Universal Robots URScript: 00B_04_Qu_BoXian.script

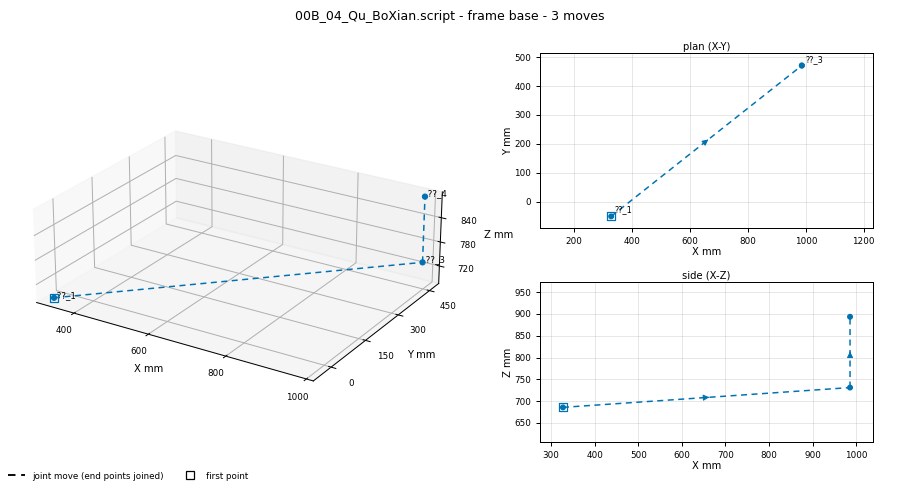
[picture p0: tool path of 00B_04_Qu_BoXian.script in frame base, 3 of 3 moves have a stored position in this frame; points joined in program order, loops and branches not executed]
def P00B_04_Qu_BoXian():
  set_gravity([0.0, 0.0, 9.82])
  set_safety_mode_transition_hardness(1)
  set_standard_analog_input_domain(0, 1)
  set_standard_analog_input_domain(1, 1)
  set_tool_analog_input_domain(0, 1)
  set_tool_analog_input_domain(1, 1)
  set_analog_outputdomain(0, 0)
  set_analog_outputdomain(1, 0)
  set_tool_voltage(24)
  set_input_actions_to_default()
  set_tcp(p[0.0,0.0,0.32,0.0,0.0,-0.5236])
  set_payload(8.0)
  global Zhua_1=[0.08063, -2.42649, -1.72682, -0.47876, 0.40808, -1.10831]
  global prepose=p[0.98979, -0.16931, -0.39963, 1.98720, 0.07234, 0.05469]
  global i_var_2=0
  global i_var_1=True
  global pose=p[0.98979, -0.31931, -0.39963, 1.98720, 0.07234, 0.05469]
  $ 1 "机器人程序"
  $ 2 "MoveJ"
  $ 3 "路点_1"
  set_tcp(p[0.0,0.0,0.32,0.0,0.0,-0.5236])
  movej(get_inverse_kin(p[.327356731489, -.050164964929, .685643613987, -.037534611162, .083188775379, 1.218470868560], qnear=[0.27391108870506287, -1.1727593580829065, -2.76978570619692, -0.833592716847555, -1.6335652510272425, -0.10533124605287725]), a=0.6981317007977318, v=0.5235987755982988)
  $ 4 "路点_3"
  set_tcp(p[0.0,0.0,0.32,0.0,0.0,-0.5236])
  movej(get_inverse_kin(p[.985999520487, .470919476195, .731087278405, .023288032010, .053106467472, 1.539289877572], qnear=[0.5973503589630127, -2.338327709828512, -1.2396519819842737, -1.1867340246783655, -1.5724447409259241, -0.10541788682045751]), a=0.6981317007977318, v=0.5235987755982988)
  $ 5 "路点_4"
  set_tcp(p[0.0,0.0,0.32,0.0,0.0,-0.5236])
  movej(get_inverse_kin(p[.985998558559, .470903374939, .893513152014, .023217172961, .053146911564, 1.539195374653], qnear=[0.5973503589630127, -2.2468321959124964, -1.0992711226092737, -1.4186251799212855, -1.572995964680807, -0.10805398622621709]), a=0.6981317007977318, v=0.5235987755982988)
end
